FUNCTION_BLOCK PUBLIC FB_SerialCommunicationRS232 EXTENDS FB_SerialCommunication
VAR_INPUT
END_VAR
VAR_OUTPUT
END_VAR
VAR
	nInternalBaudrate	:	UDINT;
END_VAR

METHOD FB_init : BOOL
VAR_INPUT
	bInitRetains	: BOOL; // if TRUE, the retain variables are initialized (warm start / cold start)
	bInCopyCode		: BOOL; // if TRUE, the instance afterwards gets moved into the copy code (online change)
	nDatabits    	: BYTE(7..8);
	eParity         : E_Parity;
	nStopbits		: BYTE(1..2);
	nBaudrate		: UDINT;	
END_VAR
THIS^.nInternalBaudrate := nBaudrate;
END_METHOD

END_FUNCTION_BLOCK

(* stored: Version 1.1.0.1, ProductVersion 3.1.4024.0
   POU FB_SerialCommunicationRS232: Id {c9884d88-d65c-4447-a13f-4478b554a409}, SpecialFunc None
   Method FB_init: Id {86750ea7-a104-44b3-9fe4-803c5400800a} *)
